Universal Robots URScript: spiral.script

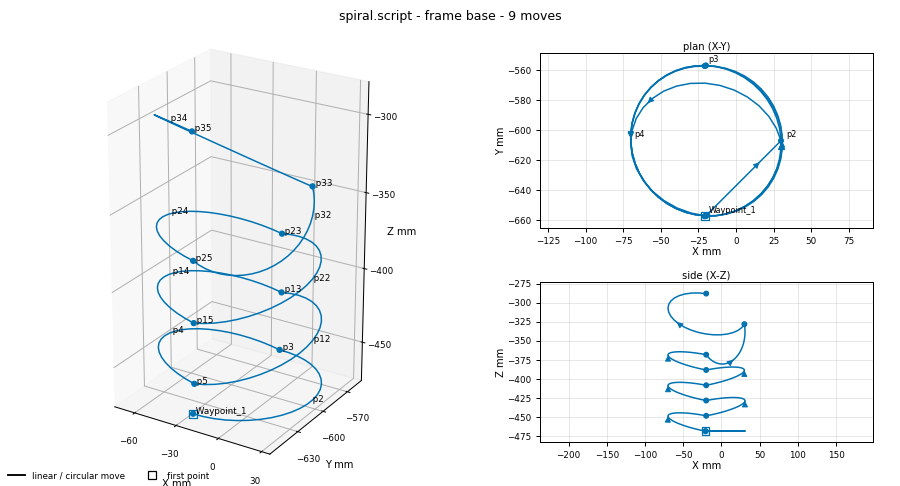
[picture p0: tool path of spiral.script in frame base, 9 of 9 moves have a stored position in this frame; points joined in program order, loops and branches not executed]
def spiral():
  global _hidden_verificationVariable=0
  set_gravity([0.0, 0.0, 9.82])
  set_target_payload(0.200000, [0.000000, 0.000000, 0.000000], [0.000105, 0.000105, 0.000105, 0.000000, 0.000000, 0.000000])
  set_tool_communication(False, 115200, 0, 1, 1.5, 3.5)
  set_tool_output_mode(0)
  set_tool_digital_output_mode(0, 2)
  set_tool_digital_output_mode(1, 1)
  set_tool_voltage(24)
  set_standard_analog_input_domain(0, 1)
  set_standard_analog_input_domain(1, 1)
  set_tool_analog_input_domain(0, 1)
  set_tool_analog_input_domain(1, 1)
  set_analog_outputdomain(0, 0)
  set_analog_outputdomain(1, 0)
  set_input_actions_to_default()
  set_safety_mode_transition_hardness(1)
  set_tcp(p[0.0,0.0,0.0,0.0,0.0,0.0])
  step_count_22ea2f5f_55fc_4f8b_8d84_b1e24e8662b1 = 0.0
  thread Step_Counter_Thread_0200fd6c_b29a_4411_9acf_5d7541d58c78():
    while (True):
      step_count_22ea2f5f_55fc_4f8b_8d84_b1e24e8662b1 = step_count_22ea2f5f_55fc_4f8b_8d84_b1e24e8662b1 + 1.0
      sync()
    end
  end
  run Step_Counter_Thread_0200fd6c_b29a_4411_9acf_5d7541d58c78()
  global Waypoint_1_p=p[-.020867848164, -.657352079433, -.468155851352, -.001221359682, 3.116276528480, .038891915640]
  global Waypoint_1_q=[-1.3400696005546742, -3.086778907952098, -1.7913300852134242, 0.14714008657437438, 1.6009042253761079, 0.22966313770202618]
  global p2_p=p[.030869999705, -.607350000191, -.468155851352, -.001221359682, 3.116276528480, .038891915640]
  global p2_q=[-1.2359479429569848, -3.105855673921777, -1.8659172948446558, 0.2440344748078682, 1.6026721347650126, 0.33381986115027984]
  global p3_p=p[-.020870000069, -.557349999933, -.468155851352, -.001221359682, 3.116276528480, .038891915640]
  global p3_q=[-1.297454072410276, -3.132935519415526, -1.9359596637680099, 0.3392260141042463, 1.6016683990903722, 0.27229163084821423]
  global p4_p=p[-.070000000057, -.607350000051, -.447999999989, -.001221359682, 3.116276528480, .038891915640]
  global p4_q=[-1.402433197750958, -3.069761714364276, -1.8928619669946052, 0.22981428723100492, 1.599687807054154, 0.16728425218790643]
  global p5_p=p[-.020000000363, -.656999999785, -.447999999959, -.001221359682, 3.116276528480, .038891915640]
  global p5_q=[-1.3386170314866952, -3.0535171607159053, -1.8227152671112439, 0.14530728032422924, 1.6009311806784563, 0.23111611573575463]
  global p12_p=p[.030869999654, -.607350000240, -.427999999944, -.001221359682, 3.116276528480, .038891915640]
  global p12_q=[-1.2359479430526088, -3.0389287679894785, -1.9277160770492703, 0.2389063510771211, 1.6026721347635535, 0.33381986105462397]
  global p13_p=p[-.020000000316, -.556999999687, -.427999999944, -.001221359682, 3.116276528480, .038891915640]
  global p13_q=[-1.2957044234606112, -3.0665522867126067, -1.9999258904475923, 0.3368630589373546, 1.6016985845798168, 0.2740418541990559]
  global p14_p=p[-.070000000069, -.607350000239, -.408000001030, -.001221359765, 3.116276528477, .038891915610]
  global p14_q=[-1.4024331978091862, -3.002302019026192, -1.9524663823080912, 0.2219590072230121, 1.599687807052194, 0.16728425207662337]
  global p15_p=p[-.020000000107, -.656999999893, -.408000001030, -.001221359765, 3.116276528477, .038891915610]
  global p15_q=[-1.338617031121986, -2.9864153794874317, -1.8809791959081306, 0.13646942792183375, 1.600931180683292, 0.2311161160475446]
  global p22_p=p[.029999999907, -.607000000093, -.388000000037, -.001221359765, 3.116276528477, .038891915610]
  global p22_q=[-1.2371558287943714, -2.9707900587303677, -1.9863144595428697, 0.22932752471465132, 1.602653571777942, 0.3326115044312951]
  global p23_p=p[-.019999999940, -.557000000060, -.388000000037, -.001221359765, 3.116276528477, .038891915610]
  global p23_q=[-1.295704422955266, -2.9981246385276754, -2.059841153956606, 0.3283506742952127, 1.6016985845858358, 0.27404185465155456]
  global p24_p=p[-.069999999907, -.606999999907, -.368000000037, -.001221359765, 3.116276528477, .038891915610]
  global p24_q=[-1.4023336331495155, -2.9332320115739314, -2.009019779799635, 0.2094452741348302, 1.5996898399193433, 0.1673838375439494]
  global p25_p=p[-.020000000060, -.656999999940, -.368000000037, -.001221359765, 3.116276528477, .038891915610]
  global p25_q=[-1.3386170310535812, -2.9179724701035963, -1.9354586232085076, 0.12250594584046157, 1.6009311806846305, 0.2311161161159622]
  global p32_p=p[.029999999907, -.607000000093, -.348000000037, -.001221359765, 3.116276528477, .038891915610]
  global p32_q=[-1.2371558287803648, -2.9005411867620614, -2.0407260959896956, 0.21349028919364468, 1.6026535717782313, 0.3326115044453072]
  global p33_p=p[.029999999833, -.607000000019, -.328000001030, -.001221359765, 3.116276528477, .038891915610]
  global p33_q=[-1.23715582885138, -2.864602806695353, -2.0665447714366083, 0.20337058457160018, 1.6026535717771653, 0.33261150437427406]
  global p34_p=p[-.070000000133, -.607000000019, -.307999999973, -.001221359765, 3.116276528477, .038891915610]
  global p34_q=[-1.4023336335373475, -2.8254877620489394, -2.0861327087458914, 0.1788139535448988, 1.599689839911492, 0.16738383715604174]
  global p35_p=p[-.020000000093, -.656999999907, -.288000000037, -.001221359765, 3.116276528477, .038891915610]
  global p35_q=[-1.3386170310660184, -2.7762840527581942, -2.0327847785438147, 0.07814368383001002, 1.6009311806844866, 0.23111611610352942]
  while (True):
    $ 1 "Robot Program"
    $ 2 "MoveP"
    $ 3 "Waypoint_1" "breakAfter"
    movep(Waypoint_1_p, a=0.25, v=0.25, r=0.025)
    $ 4 "CircleMove"
    $ 5 "p2" "noBreak"
    $ 6 "p3" "breakAfter"
    movec(p2_p, p3_p, a=0.25, v=0.25, r=0.025)
    $ 7 "CircleMove"
    $ 8 "p4" "noBreak"
    $ 9 "p5" "breakAfter"
    movec(p4_p, p5_p, a=1.2, v=0.25, r=0.025)
    $ 10 "CircleMove"
    $ 11 "p12" "noBreak"
    $ 12 "p13" "breakAfter"
    movec(p12_p, p13_p, a=1.2, v=0.25, r=0.025)
    $ 13 "CircleMove"
    $ 14 "p14" "noBreak"
    $ 15 "p15" "breakAfter"
    movec(p14_p, p15_p, a=1.2, v=0.25, r=0.025)
    $ 16 "CircleMove"
    $ 17 "p22" "noBreak"
    $ 18 "p23" "breakAfter"
    movec(p22_p, p23_p, a=1.2, v=0.25, r=0.025)
    $ 19 "CircleMove"
    $ 20 "p24" "noBreak"
    $ 21 "p25" "breakAfter"
    movec(p24_p, p25_p, a=1.2, v=0.25, r=0.025)
    $ 22 "CircleMove"
    $ 23 "p32" "noBreak"
    $ 24 "p33" "breakAfter"
    movec(p32_p, p33_p, a=1.2, v=0.25, r=0.025)
    $ 25 "CircleMove"
    $ 26 "p34" "noBreak"
    $ 27 "p35" "breakAfter"
    movec(p34_p, p35_p, a=1.2, v=0.25, r=0.025)
  end
end
